{region '#Template'}
	{attribute 'Version' := '5.0.0.0'}
	{attribute 'Tags' := '"LCID": "1031", "Text": "General, Cabinet, Control cabinet, Event groups, Categories, Notification classes, Event classes"'}
	{attribute 'Tags' := '"LCID": "1033", "Text": "General, Cabinet, Control cabinet, Event groups, Categories, Notification classes, Event classes"'}
	{attribute 'Using' := '"Type": "Template", "URI": "EC_ID"'}
	{attribute 'Description' := '"LCID": "1031", "Text": "Ereignisgruppen, Kategorien"'}
	{attribute 'Description' := '"LCID": "1033", "Text": "Event groups, categories"'}
{endregion}
FUNCTION_BLOCK FB_BA_EvtGroups EXTENDS FB_BA_View
VAR_INPUT CONSTANT
	LifeSafety						: FB_BA_EvtCategory;
	SafetyMsg						: FB_BA_EvtCategory;
	AlarmMsg						: FB_BA_EvtCategory;
	FaultMsg						: FB_BA_EvtCategory;
	MaintenanceMsg01				: FB_BA_EvtCategory;
	MaintenanceMsg02				: FB_BA_EvtCategory;
	SystemMsg						: FB_BA_EvtCategory;
	ManualOp						: FB_BA_EvtCategory;
	OtherMsg						: FB_BA_EvtCategory;
END_VAR

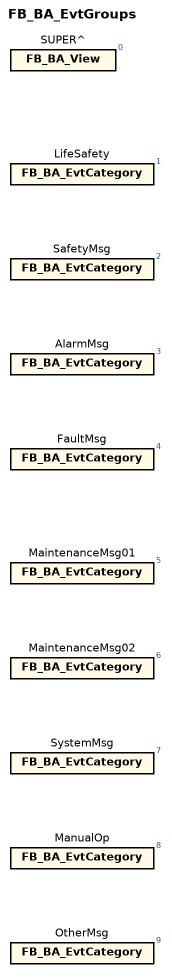
SUPER^(); // FB_BA_View
LifeSafety(); // FB_BA_EvtCategory
SafetyMsg(); // FB_BA_EvtCategory
AlarmMsg(); // FB_BA_EvtCategory
FaultMsg(); // FB_BA_EvtCategory
MaintenanceMsg01(); // FB_BA_EvtCategory
MaintenanceMsg02(); // FB_BA_EvtCategory
SystemMsg(); // FB_BA_EvtCategory
ManualOp(); // FB_BA_EvtCategory
OtherMsg(); // FB_BA_EvtCategory

METHOD FB_init : BOOL
VAR_INPUT
	bInitRetains : BOOL; // if TRUE, the retain variables are initialized (warm start / cold start)
	bInCopyCode : BOOL;  // if TRUE, the instance afterwards gets moved into the copy code (online change)
END_VAR
//===================================================================
// Ereigniskategorie - Gefahr für Leben // Event category - Danger to life
// Brandalarm, Überfall // Fire alarm, robbery
LifeSafety.iParent							:= THIS^;
LifeSafety.iLabel							:= LblCtl_EvtCategoryLifeSafty;
LifeSafety.eDPADMode						:= E_BA_DPADMode.eInclude;																						
LifeSafety.EC.nInstanceID					:= EC_ID.NC10;
LifeSafety.EC.iLabel						:= LblFun_ObjectNotificationClass;
LifeSafety.EC.sObjectName					:='{Idx=10}';
LifeSafety.EC.eAlarmMode					:= E_BA_AlarmMode.UserDefined;
LifeSafety.EC.eEventType					:= E_BA_EventType.eAlarm;
LifeSafety.EC.aPriority[1]					:= 10;
LifeSafety.EC.aPriority[2]					:= 11;
LifeSafety.EC.aPriority[3]					:= 12;
LifeSafety.EC.aAcknowledgeRequired[1]		:= TRUE;
LifeSafety.EC.aAcknowledgeRequired[2]		:= FALSE;
LifeSafety.EC.aAcknowledgeRequired[3]		:= TRUE;
//===================================================================		
// Ereigniskategorie - Gefahrenmeldung, Sicherheitsmeldung // Event category - hazard alert, safety message
// Einbruch, unberechtigter Zutritt // Burglary, unauthorised entry
SafetyMsg.iParent							:= THIS^;
SafetyMsg.iLabel							:= LblCtl_EvtCategorySaftyMessage;
SafetyMsg.eDPADMode							:= E_BA_DPADMode.eInclude;																						
SafetyMsg.EC.nInstanceID					:= EC_ID.NC20;
SafetyMsg.EC.iLabel							:= LblFun_ObjectNotificationClass;
SafetyMsg.EC.sObjectName					:='{Idx=20}';
SafetyMsg.EC.eAlarmMode						:= E_BA_AlarmMode.UserDefined;
SafetyMsg.EC.eEventType						:= E_BA_EventType.eAlarm;
SafetyMsg.EC.aPriority[1]					:= 40;
SafetyMsg.EC.aPriority[2]					:= 41;
SafetyMsg.EC.aPriority[3]					:= 42;
SafetyMsg.EC.aAcknowledgeRequired[1]		:= TRUE;
SafetyMsg.EC.aAcknowledgeRequired[2]		:= FALSE;
SafetyMsg.EC.aAcknowledgeRequired[3]		:= TRUE;
//===================================================================//
// Ereigniskategorie - Alarmeldung - Meldung signalisiert Anlagenausfall oder erfordert sofortigen Eingriff 
// Event category - Alarm message - Message signals system failure or requires immediate intervention 
// Sicherheitstemperaturbegrenzer (STB), Sicherheitsdruckbegrenzer (SDB), Übertemperatur der Warmwasserbereitung (WWB), Sicherheitsventile, Hauptpumpen, Keilriemenwächter, Frequenzumformer, Kälteanlagen, Spannungsausfall usw
// Safety temperature limiter, safety pressure limiter, excess temperature of water heating, safety valves, main pumps, V-belt monitors, frequency converters, refrigeration systems, voltage failure, etc.
AlarmMsg.iParent							:= THIS^;
AlarmMsg.iLabel								:= LblCtl_EvtCategoryAlarmMessage;
AlarmMsg.eDPADMode							:= E_BA_DPADMode.eInclude;																						
AlarmMsg.EC.nInstanceID						:= EC_ID.NC30;
AlarmMsg.EC.iLabel							:= LblFun_ObjectNotificationClass;
AlarmMsg.EC.sObjectName						:= '{Idx=30}'	;
AlarmMsg.EC.eAlarmMode						:= E_BA_AlarmMode.UserDefined;
AlarmMsg.EC.eEventType						:= E_BA_EventType.eAlarm;
AlarmMsg.EC.aPriority[1]					:= 70;
AlarmMsg.EC.aPriority[2]					:= 71;
AlarmMsg.EC.aPriority[3]					:= 72;
AlarmMsg.EC.aAcknowledgeRequired[1]			:= TRUE;
AlarmMsg.EC.aAcknowledgeRequired[2]			:= FALSE;
AlarmMsg.EC.aAcknowledgeRequired[3]			:= TRUE;

//===================================================================
// Ereigniskategorie - Störungsmeldung - Meldung weist auf einen anormalen Betriebszustand hin
// Event category - malfunction message - message indicates abnormal operating condition
// Temperaturwächter (TW), Druckwächter (DW), Temperaturüberwachung von Wärmetauscher (WT) und WWB, Motorschutz, Aufzug-Sammelstörmeldung, Netzdrücke usw.
// Temperature monitor, pressure monitor, temperature monitoring of heat exchanger and water heating, motor protection, lift collective fault signal, mains pressures, etc.
FaultMsg.iParent							:= THIS^;
FaultMsg.iLabel								:= LblCtl_EvtCategoryFaultMessage;
FaultMsg.eDPADMode							:= E_BA_DPADMode.eInclude;																						
FaultMsg.EC.nInstanceID						:= EC_ID.NC40;
FaultMsg.EC.iLabel							:= LblFun_ObjectNotificationClass;
FaultMsg.EC.sObjectName						:= '{Idx=40}'	;
FaultMsg.EC.eAlarmMode						:= E_BA_AlarmMode.UserDefined;
FaultMsg.EC.eEventType						:= E_BA_EventType.eDisturb;
FaultMsg.EC.aPriority[1]					:= 100;
FaultMsg.EC.aPriority[2]					:= 101;
FaultMsg.EC.aPriority[3]					:= 102;
FaultMsg.EC.aAcknowledgeRequired[1]			:= TRUE;
FaultMsg.EC.aAcknowledgeRequired[2]			:= FALSE;
FaultMsg.EC.aAcknowledgeRequired[3]			:= FALSE;
//===================================================================
// Ereigniskategorie - Wartungsmeldung, Hinweis auf Wartungsaktivität o.ä.
// Event category - Maintenance message Maintenance message, indication of maintenance activity or similar.
// Betriebsstunden, Behälterstand, Reparaturschalter usw.
// Operating hours, tank level, repair switch, etc.
MaintenanceMsg01.iParent					:= THIS^;
MaintenanceMsg01.iLabel						:= LblCtl_EvtCategoryMaintenanceMessage;
MaintenanceMsg01.eDPADMode					:= E_BA_DPADMode.eInclude;																						
MaintenanceMsg01.EC.nInstanceID				:= EC_ID.NC50;
MaintenanceMsg01.EC.iLabel					:= LblFun_ObjectNotificationClass;
MaintenanceMsg01.EC.sObjectName				:= '{Idx=50}'	;
MaintenanceMsg01.EC.eAlarmMode				:= E_BA_AlarmMode.UserDefined;
MaintenanceMsg01.EC.eEventType				:= E_BA_EventType.eMaintenance;
MaintenanceMsg01.EC.aPriority[1]			:= 130;
MaintenanceMsg01.EC.aPriority[2]			:= 131;
MaintenanceMsg01.EC.aPriority[3]			:= 132;
MaintenanceMsg01.EC.aAcknowledgeRequired[1]	:= TRUE;
MaintenanceMsg01.EC.aAcknowledgeRequired[2]	:= FALSE;
MaintenanceMsg01.EC.aAcknowledgeRequired[3]	:= FALSE;

// Filterende erreicht, Filter verschmutzt usw.
// Filter end reached, filter dirty, etc.
MaintenanceMsg02.iParent					:= THIS^;
MaintenanceMsg02.iLabel						:= LblCtl_EvtCategoryMaintenanceMessage;
MaintenanceMsg02.eDPADMode					:= E_BA_DPADMode.eInclude;																						
MaintenanceMsg02.EC.nInstanceID				:= EC_ID.NC51;
MaintenanceMsg02.EC.iLabel					:= LblFun_ObjectNotificationClass;
MaintenanceMsg02.EC.sObjectName				:= '{Idx=51}'	;
MaintenanceMsg02.EC.eAlarmMode				:= E_BA_AlarmMode.UserDefined;
MaintenanceMsg02.EC.eEventType				:= E_BA_EventType.eMaintenance;
MaintenanceMsg02.EC.aPriority[1]			:= 135;
MaintenanceMsg02.EC.aPriority[2]			:= 136;
MaintenanceMsg02.EC.aPriority[3]			:= 137;
MaintenanceMsg02.EC.aAcknowledgeRequired[1]	:= TRUE;
MaintenanceMsg02.EC.aAcknowledgeRequired[2]	:= FALSE;
MaintenanceMsg02.EC.aAcknowledgeRequired[3]	:= FALSE;
//===================================================================
//===================================================================
// Ereigniskategorie - Systemmeldung, Störungsmeldung aus GA-System
// Event category - System message, System message, Fault message from building automation system
// Gerätestörung, Batteriemeldung, Kommunikationsunterbrechung usw.
// Unit malfunction, battery message, communication interruption, etc.
SystemMsg.iParent							:= THIS^;
SystemMsg.iLabel							:= LblCtl_EvtCategorySystem;
SystemMsg.eDPADMode							:= E_BA_DPADMode.eInclude;																						
SystemMsg.EC.nInstanceID					:= EC_ID.NC60;
SystemMsg.EC.iLabel							:= LblFun_ObjectNotificationClass;
SystemMsg.EC.sObjectName					:='{Idx=60}';
SystemMsg.EC.eAlarmMode						:= E_BA_AlarmMode.UserDefined;
SystemMsg.EC.eEventType						:= E_BA_EventType.eNotification;
SystemMsg.EC.aPriority[1]					:= 180;
SystemMsg.EC.aPriority[2]					:= 181;
SystemMsg.EC.aPriority[3]					:= 182;
SystemMsg.EC.aAcknowledgeRequired[1]		:= FALSE;
SystemMsg.EC.aAcknowledgeRequired[2]		:= FALSE;
SystemMsg.EC.aAcknowledgeRequired[3]		:= FALSE;
//===================================================================//
//	Ereigniskategorie - Manual operation, Handeingriff
ManualOp.iParent							:= THIS^;
ManualOp.iLabel								:= LblCtl_EvtCategoryManualOperation;
ManualOp.eDPADMode							:= E_BA_DPADMode.eInclude;																						
ManualOp.EC.nInstanceID						:= EC_ID.NC70;
ManualOp.EC.iLabel							:= LblFun_ObjectNotificationClass;
ManualOp.EC.sObjectName						:='{Idx=70}';
ManualOp.EC.eAlarmMode						:= E_BA_AlarmMode.UserDefined;
ManualOp.EC.eEventType						:= E_BA_EventType.eOther;
ManualOp.EC.aPriority[1]					:= 220;
ManualOp.EC.aPriority[2]					:= 220;
ManualOp.EC.aPriority[3]					:= 220;
ManualOp.EC.aAcknowledgeRequired[1]			:= FALSE;
ManualOp.EC.aAcknowledgeRequired[2]			:= FALSE;
ManualOp.EC.aAcknowledgeRequired[3]			:= FALSE;
//===================================================================//
// Ereigniskategorie - Freibleibend, Sonstige Meldungen
// Event category - Other message, Not binding, Other messages
// Betriebszustandswechsel, Betriebsarten, Trendspeicher voll usw.
// Operating status change, operating modes, trend memory full, etc.
OtherMsg.iParent							:= THIS^;
OtherMsg.iLabel								:= LblCtl_EvtCategoryOther;
OtherMsg.eDPADMode							:= E_BA_DPADMode.eInclude;																						
OtherMsg.EC.nInstanceID						:= EC_ID.NC80;
OtherMsg.EC.iLabel							:= LblFun_ObjectNotificationClass;
OtherMsg.EC.sObjectName						:='{Idx=80}';
OtherMsg.EC.eAlarmMode						:= E_BA_AlarmMode.UserDefined;
OtherMsg.EC.eEventType						:= E_BA_EventType.eOther;
OtherMsg.EC.aPriority[1]					:= 230;
OtherMsg.EC.aPriority[2]					:= 231;
OtherMsg.EC.aPriority[3]					:= 232;
OtherMsg.EC.aAcknowledgeRequired[1]			:= FALSE;
OtherMsg.EC.aAcknowledgeRequired[2]			:= FALSE;
OtherMsg.EC.aAcknowledgeRequired[3]			:= FALSE;
END_METHOD

END_FUNCTION_BLOCK

(* stored: Version 1.1.0.1, ProductVersion 3.1.4024.12
   POU FB_BA_EvtGroups: Id {fff5eac5-352b-4cd3-98f5-1dc2f4290163}, SpecialFunc None
   Method FB_init: Id {5327786a-2cda-4494-ad0f-329f7ea9cacc} *)
